{attribute 'qualified_only'}
VAR_GLOBAL
	(* Digital IO to Byte *)
	aDigitalInputIO AT %I* 	: ARRAY[1..9]OF BYTE; //KL1408 9EA
	aDigitalOutputIO AT %Q* : ARRAY[1..4]OF BYTE; //KL2408 4EA
	
	(* Analog Input to INT*)
	aAnalogInputIO AT %I* 	: ARRAY[1..40]OF INT;
	aAnalogOutputIO AT %Q* 	: ARRAY[1..29]OF INT;
	aAnalogInputIO2 AT %I*	: ARRAY[1..2]OF UINT;
	
	(*Solenoid Valve*)
	aOutputSolValve AT %Q* 	: ARRAY[1..3]OF DWORD; //Solenoid Valve
	
	(* Read and Write of Device Control Value*)
	aMaxValueController		: ARRAY[1..29]OF REAL ; //Device Max Value from UI
	aController 			: ARRAY[1..29] OF FB_RampGenerator; //MFC, EPC 0 ~ 5V
	aController_TV 			: ARRAY[1..29] OF REAL; //Target Value from UI
	aController_RampTime 	: ARRAY[1..29] OF INT;
	aController_PV 			: ARRAY[1..29] OF REAL; //Present Value from Device
	aController_CV 			: ARRAY[1..29] OF REAL; //Current Value from RampingController
	
	(* Present Value Meter Display*)
	aMonitoring_PV 			: ARRAY[1..17] OF REAL; //Gauge Monitoring Value to UI
	aInputState				: ARRAY[1..5] OF WORD; // Digital Input from Device (Switch)
	aOutputCmd				: ARRAY[1..3] OF WORD; // Digital Command from UI
	aInterlock				: ARRAY[1..5] OF DWORD; // Interlock
	aInterlockSet			: ARRAY[1..16] OF REAL; // UI Interlokc Setting Value
	aInterlockEnable		: ARRAY[1..6] OF DWORD; // UI Interlock Enable Setting
	
	nCaseSignalTower		: INT;
	nDorOperationError		: INT;
	bDorState				: BOOL;
	bDorOnEnable			: BOOL;
// 	bE3508_HeaterOn			: BOOL;
	wE3508_CV				: WORD;
	wE3508_PV				: WORD;
	wIqPlus_CV				: WORD;
	wIqPlus_CDG1_PV			: WORD;
	wIqPlus_CDG2_PV			: WORD;
	nRotation_Converted_PV	: INT;
	rRotation_ControlValue	: REAL;
	nIQPLUS_SetType 		: INT;
	nIQPLUS_Mode			: INT;
	aLineHeater_rTemperaturePV : ARRAY[1..8]OF REAL;
	nE3508_nInputManAutoBytes : USINT;
	isCoverClosed 			: BOOL;
	isPumpRunning 			: BOOL;
END_VAR

VAR_GLOBAL CONSTANT
	KL3464MaxValueH	: REAL := 16383; //0~5V Half Input
	KL3464MaxValue 	: REAL := 32767; //0~10V
	KL4404MaxValueH	: REAL := 16383; //0~5V Half Output
	KL3054MaxValue 	: REAL := 32767; //4~20mA
	KL3152MaxValue	: REAL := 65535; //4~20mA
	KL3204MaxValue 	: REAL := 32767; //4~20mA
END_VAR

(* stored: Version 1.1.0.1, ProductVersion 3.1.4026.11
   GVL GVL_IO: Id {a5f3292d-798a-4b6c-af88-b59309d83086} *)
